KUKA KRL program: EOAChangerControl.src, EOAChangerControl.dat

--- EOAChangerControl.src ---
&ACCESS RVO4
&REL 10
&PARAM DISKPATH = KRC:\R1\TP\CNCR TP\Schunk
DEF EOAChangerControl( )

;************************************************
;              CNC Robotics Ltd
;              www.cncrobotics.co.uk
;************************************************
;     Contact: helpdesk@cncrobotics.co.uk
;     Date: 25/09/23
;     Version: 0.14.46
;************************************************
; Description: Programs for swapping the EOA tool.
;************************************************

END

GLOBAL DEF SwapTool(newTool:IN)
DECL EOA_TOOL_TYPE newTool
;HomeRobot()

HomePosition()
;WAIT FOR NOT iEOAFault
DropEOATool(ToolOnRobot)
WAIT SEC 0
nSchunkOKSwapAns = 0

WHILE nSchunkOKSwapAns<>1

MsgDialog(nSchunkOKSwapAns,"Swap the tool balance clips to the new tool","Schunk",,,,,,,"Cancel","Continue", FALSE, nSchunkMsg, E_spsMsgOpt)

ENDWHILE

PickUpEOATool(newTool)

HomePosition()
END

GLOBAL DEF DropEOATool(tool:IN)
DECL EOA_TOOL_TYPE tool

;WAIT FOR NOT iEOAFault

SWITCH tool
   CASE #SPINDLE

      IF nToolHeld <> 0 THEN
         ToolCheck()
      ELSE
         WAIT FOR (nToolHeld == 0) AND (NOT iToolLocked)
      ENDIF
      ToolRackClose()
      DropSpindle()
      bToolOnRobot = FALSE

   CASE #CEAD

      DropCead()
      bToolOnRobot = FALSE

   CASE #NONE
      EOAChangeSafe()
     ; WAIT FOR iEOALocked AND NOT iEOAUnlocked
      bToolOnRobot = FALSE
ENDSWITCH

END

GLOBAL DEF PickupEOATool(tool:IN)
DECL EOA_TOOL_TYPE tool

IF tool == #NONE THEN
   RETURN
ENDIF


EOAChangeSafe()

WAIT FOR NOT (iSpindleOnRobot OR iCeadOnRobot)

SWITCH tool
   CASE #SPINDLE
      ;Move to spindle pick position
      PickUpSpindle()
      bToolOnRobot = TRUE
   CASE #CEAD

      ;Move to Extruder pick position
      PickUpCEAD()
      ;halt
      WAIT FOR iCeadOnRobot
      IF NOT iNoEmergency THEN
         PULSE(oAckErrors,TRUE,1)
      ENDIF
      bToolOnRobot = TRUE
      ;Retract extruder from post

      ;halt
   CASE #NONE

ENDSWITCH
EOAChangeSafe()


END

GLOBAL DEF LockEOAChanger(tool:IN)
DECL EOA_TOOL_TYPE tool

WAIT FOR iAirOk

oEOAUnlock = FALSE
oEOANotLock = FALSE

WAIT FOR NOT iEOAUnlocked

IF tool <> #NONE THEN
   WAIT FOR iEOALocked
ENDIF

IF tool == #CEAD THEN
   WAIT FOR iCeadOnRobot
      IF NOT iNoEmergency THEN
         PULSE(oAckErrors,TRUE,1)
      ENDIF
ENDIF

bToolOnRobot = TRUE AND (tool <> #NONE)
toolOnRobot = tool

WAIT SEC 1

END

GLOBAL DEF UnlockEOAChanger()

WAIT FOR iAirOk

bToolOnRobot = FALSE

oEOANotLock = TRUE
oEOAUnlock = TRUE

WAIT FOR iEOAUnlocked AND NOT iEOALocked

toolOnRobot = #NONE

WAIT SEC 1

END

GLOBAL DEF SetNullTool(tool:IN)
DECL EOA_TOOL_TYPE tool

Switch tool
   CASE #SPINDLE
      BAS(#TOOL, 31)
   CASE #CEAD
      BAS(#TOOL, 32)
   CASE #NONE
      BAS(#TOOL, 0)
ENDSWITCH

END


GLOBAL DEF NullPTP(tool:IN, MoveTo:IN)
DECL EOA_TOOL_TYPE tool
DECL E6POS MoveTo

BAS(#BASE, 0)

SetNullTool(tool)


BAS(#VEL_PTP,20)


PTP MoveTo

END

GLOBAL DEFFCT BOOL CheckEOAinputs (tool:IN)
DECL EOA_TOOL_TYPE tool

SWITCH tool
CASE #SPINDLE
   RETURN iSpindleOnRobot
CASE #CEAD
   RETURN iCeadOnRobot
CASE #NONE
   RETURN NOT(iCeadOnRobot OR iSpindleOnRobot)
ENDSWITCH


ENDFCT

GLOBAL DEF CheckEOATooling(tool:IN)
DECL INT _nAns
DECL EOA_TOOL_TYPE tool

_nAns = 0

WHILE ( (CheckEOAinputs(tool)) AND (toolOnRobot<>tool) )

MsgDialog(_nAns,"Incorrect EOA tooling. Cancel program and change EOA tooling","Schunk",,,,,,,,"Cancel", FALSE, nSchunkMsg, E_spsMsgOpt)

ENDWHILE

END

--- EOAChangerControl.dat ---
&ACCESS  RV
&PARAM DISKPATH = KRC:\R1\TP\CNCR TP\Schunk
&REL 9
DEFDAT  EOACHANGERCONTROL PUBLIC

;Global Variables
GLOBAL BOOL bToolOnRobot=TRUE
GLOBAL BOOL bSchunkFault=FALSE
GLOBAL ENUM EOA_TOOL_TYPE CEAD,SPINDLE,NONE
DECL GLOBAL EOA_TOOL_TYPE toolOnRobot=#SPINDLE
GLOBAL INT nSchunkOKSwapAns=1

DECL BASIS_SUGG_T LAST_BASIS={POINT1[] "P18                     ",POINT2[] "P18                     ",CP_PARAMS[] "CPDAT18                 ",PTP_PARAMS[] "PDAT0                   ",CONT[] "                        ",CP_VEL[] "0.05                    ",PTP_VEL[] "100                     ",SYNC_PARAMS[] "SYNCDAT                 ",SPL_NAME[] "S0                      ",A_PARAMS[] "ADAT0                   "}
DECL E6POS XP1={X 2110.28467,Y 207.085190,Z 2.20077252,A 89.6821136,B 59.9209824,C 90.9203,S 22,T 59,E1 -360.000763,E2 0.0,E3 0.0,E4 0.0,E5 0.0,E6 0.0}
DECL FDAT FP1={TOOL_NO 0,BASE_NO 0,IPO_FRAME #BASE,POINT2[] " ",TQ_STATE FALSE}
DECL LDAT LCPDAT1={VEL 2.00000,ACC 100.000,APO_DIST 100.000,APO_FAC 50.0000,AXIS_VEL 100.000,AXIS_ACC 100.000,ORI_TYP #VAR,CIRC_TYP #BASE,JERK_FAC 50.0000,GEAR_JERK 50.0000,EXAX_IGN 0}
DECL E6POS XP2={X 2415.83740,Y 208.572250,Z 1.01012671,A 89.8723297,B 60.1981316,C 91.1378,S 22,T 59,E1 -360.000763,E2 0.0,E3 0.0,E4 0.0,E5 0.0,E6 0.0}
DECL FDAT FP2={TOOL_NO 0,BASE_NO 0,IPO_FRAME #BASE,POINT2[] " ",TQ_STATE FALSE}
DECL LDAT LCPDAT2={VEL 2.00000,ACC 5.00000,APO_DIST 100.000,APO_FAC 50.0000,AXIS_VEL 100.000,AXIS_ACC 100.000,ORI_TYP #VAR,CIRC_TYP #BASE,JERK_FAC 50.0000,GEAR_JERK 50.0000,EXAX_IGN 0}
DECL E6POS XP3={X 2415.85522,Y 208.560196,Z 40.6353645,A 89.8745,B 60.1985,C 91.1395645,S 22,T 59,E1 -360.000763,E2 0.0,E3 0.0,E4 0.0,E5 0.0,E6 0.0}
DECL FDAT FP3={TOOL_NO 0,BASE_NO 0,IPO_FRAME #BASE,POINT2[] " ",TQ_STATE FALSE}
DECL LDAT LCPDAT3={VEL 2.00000,ACC 5.00000,APO_DIST 100.000,APO_FAC 50.0000,AXIS_VEL 100.000,AXIS_ACC 100.000,ORI_TYP #VAR,CIRC_TYP #BASE,JERK_FAC 50.0000,GEAR_JERK 50.0000,EXAX_IGN 0}
DECL E6POS XP4={X 2116.75293,Y 208.708710,Z 41.8776550,A 89.8257751,B 60.1956673,C 91.0831833,S 22,T 59,E1 -360.000763,E2 0.0,E3 0.0,E4 0.0,E5 0.0,E6 0.0}
DECL FDAT FP4={TOOL_NO 0,BASE_NO 0,IPO_FRAME #BASE,POINT2[] " ",TQ_STATE FALSE}
DECL LDAT LCPDAT4={VEL 2.00000,ACC 5.00000,APO_DIST 100.000,APO_FAC 50.0000,AXIS_VEL 100.000,AXIS_ACC 100.000,ORI_TYP #VAR,CIRC_TYP #BASE,JERK_FAC 50.0000,GEAR_JERK 50.0000,EXAX_IGN 0}
DECL E6POS XP5={X 2110.28589,Y 207.069,Z 53.0706749,A 89.6858215,B 59.9213676,C 90.9231262,S 22,T 59,E1 -360.000763,E2 0.0,E3 0.0,E4 0.0,E5 0.0,E6 0.0}
DECL FDAT FP5={TOOL_NO 0,BASE_NO 0,IPO_FRAME #BASE,POINT2[] " ",TQ_STATE FALSE}
DECL LDAT LCPDAT5={VEL 2.00000,ACC 100.000,APO_DIST 100.000,APO_FAC 50.0000,AXIS_VEL 100.000,AXIS_ACC 100.000,ORI_TYP #VAR,CIRC_TYP #BASE,JERK_FAC 50.0000,GEAR_JERK 50.0000,EXAX_IGN 0}
DECL E6POS XP6={X 2416.12964,Y 209.042725,Z 41.9984512,A 89.6551743,B 60.2458687,C 91.1575,S 22,T 59,E1 -360.000763,E2 0.0,E3 0.0,E4 0.0,E5 0.0,E6 0.0}
DECL FDAT FP6={TOOL_NO 0,BASE_NO 0,IPO_FRAME #BASE,POINT2[] " ",TQ_STATE FALSE}
DECL LDAT LCPDAT6={VEL 2.00000,ACC 5.00000,APO_DIST 100.000,APO_FAC 50.0000,AXIS_VEL 100.000,AXIS_ACC 100.000,ORI_TYP #VAR,CIRC_TYP #BASE,JERK_FAC 50.0000,GEAR_JERK 50.0000,EXAX_IGN 0}
DECL E6POS XP7={X 2416.11230,Y 209.054535,Z 3.29431415,A 89.6530533,B 60.2455025,C 91.1557693,S 22,T 59,E1 -360.000763,E2 0.0,E3 0.0,E4 0.0,E5 0.0,E6 0.0}
DECL FDAT FP7={TOOL_NO 0,BASE_NO 0,IPO_FRAME #BASE,POINT2[] " ",TQ_STATE FALSE}
DECL LDAT LCPDAT7={VEL 2.00000,ACC 5.00000,APO_DIST 100.000,APO_FAC 50.0000,AXIS_VEL 100.000,AXIS_ACC 100.000,ORI_TYP #VAR,CIRC_TYP #BASE,JERK_FAC 50.0000,GEAR_JERK 50.0000,EXAX_IGN 0}
DECL E6POS XP8={X 2412.57593,Y 209.057129,Z 1.56290293,A 89.6524,B 60.2454529,C 91.1550293,S 22,T 59,E1 -360.000763,E2 0.0,E3 0.0,E4 0.0,E5 0.0,E6 0.0}
DECL FDAT FP8={TOOL_NO 0,BASE_NO 0,IPO_FRAME #BASE,POINT2[] " ",TQ_STATE FALSE}
DECL LDAT LCPDAT8={VEL 2.00000,ACC 5.00000,APO_DIST 100.000,APO_FAC 50.0000,AXIS_VEL 100.000,AXIS_ACC 100.000,ORI_TYP #VAR,CIRC_TYP #BASE,JERK_FAC 50.0000,GEAR_JERK 50.0000,EXAX_IGN 0}
DECL E6POS XP9={X 2225.87671,Y 209.156555,Z 2.36978531,A 89.6218,B 60.2435684,C 91.1194611,S 22,T 59,E1 -360.000763,E2 0.0,E3 0.0,E4 0.0,E5 0.0,E6 0.0}
DECL FDAT FP9={TOOL_NO 0,BASE_NO 0,IPO_FRAME #BASE,POINT2[] " ",TQ_STATE FALSE}
DECL LDAT LCPDAT9={VEL 2.00000,ACC 100.000,APO_DIST 100.000,APO_FAC 50.0000,AXIS_VEL 100.000,AXIS_ACC 100.000,ORI_TYP #VAR,CIRC_TYP #BASE,JERK_FAC 50.0000,GEAR_JERK 50.0000,EXAX_IGN 0}
DECL E6POS XP10={X 2268.25537,Y 206.572342,Z 1090.06494,A 90.2147751,B 60.5988121,C 91.2159958,S 22,T 59,E1 -360.000763,E2 0.0,E3 0.0,E4 0.0,E5 0.0,E6 0.0}
DECL FDAT FP10={TOOL_NO 0,BASE_NO 0,IPO_FRAME #BASE,POINT2[] " ",TQ_STATE FALSE}
DECL LDAT LCPDAT10={VEL 2.00000,ACC 100.000,APO_DIST 100.000,APO_FAC 50.0000,AXIS_VEL 100.000,AXIS_ACC 100.000,ORI_TYP #VAR,CIRC_TYP #BASE,JERK_FAC 50.0000,GEAR_JERK 50.0000,EXAX_IGN 0}
DECL E6POS XP11={X 2441.39771,Y 206.522354,Z 1089.56934,A 90.2275467,B 60.5963249,C 91.2292,S 22,T 59,E1 -360.000763,E2 0.0,E3 0.0,E4 0.0,E5 0.0,E6 0.0}
DECL FDAT FP11={TOOL_NO 0,BASE_NO 0,IPO_FRAME #BASE,POINT2[] " ",TQ_STATE FALSE}
DECL LDAT LCPDAT11={VEL 2.00000,ACC 5.00000,APO_DIST 100.000,APO_FAC 50.0000,AXIS_VEL 100.000,AXIS_ACC 100.000,ORI_TYP #VAR,CIRC_TYP #BASE,JERK_FAC 50.0000,GEAR_JERK 50.0000,EXAX_IGN 0}
DECL E6POS XP12={X 2441.48755,Y 206.521118,Z 1137.87341,A 90.2316818,B 60.5967445,C 91.2319260,S 22,T 59,E1 -360.000763,E2 0.0,E3 0.0,E4 0.0,E5 0.0,E6 0.0}
DECL FDAT FP12={TOOL_NO 0,BASE_NO 0,IPO_FRAME #BASE,POINT2[] " ",TQ_STATE FALSE}
DECL LDAT LCPDAT12={VEL 2.00000,ACC 5.00000,APO_DIST 100.000,APO_FAC 50.0000,AXIS_VEL 100.000,AXIS_ACC 100.000,ORI_TYP #VAR,CIRC_TYP #BASE,JERK_FAC 50.0000,GEAR_JERK 50.0000,EXAX_IGN 0}
DECL E6POS XP13={X 1809.98462,Y 206.676010,Z 1139.42065,A 90.1941833,B 60.6061363,C 91.1919708,S 22,T 59,E1 -360.000763,E2 0.0,E3 0.0,E4 0.0,E5 0.0,E6 0.0}
DECL FDAT FP13={TOOL_NO 0,BASE_NO 0,IPO_FRAME #BASE,POINT2[] " ",TQ_STATE FALSE}
DECL LDAT LCPDAT13={VEL 2.00000,ACC 100.000,APO_DIST 100.000,APO_FAC 50.0000,AXIS_VEL 100.000,AXIS_ACC 100.000,ORI_TYP #VAR,CIRC_TYP #BASE,JERK_FAC 50.0000,GEAR_JERK 50.0000,EXAX_IGN 0}
DECL E6POS XP14={X 2137.01392,Y 206.603485,Z 1138.69543,A 90.2108,B 60.6013184,C 91.2106476,S 22,T 59,E1 -360.000763,E2 0.0,E3 0.0,E4 0.0,E5 0.0,E6 0.0}
DECL FDAT FP14={TOOL_NO 0,BASE_NO 0,IPO_FRAME #BASE,POINT2[] " ",TQ_STATE FALSE}
DECL LDAT LCPDAT14={VEL 2.00000,ACC 100.000,APO_DIST 100.000,APO_FAC 50.0000,AXIS_VEL 100.000,AXIS_ACC 100.000,ORI_TYP #VAR,CIRC_TYP #BASE,JERK_FAC 50.0000,GEAR_JERK 50.0000,EXAX_IGN 0}
DECL E6POS XP15={X 2441.50073,Y 206.183929,Z 1133.35229,A 90.2278366,B 60.3237762,C 91.2293854,S 22,T 59,E1 -360.000763,E2 0.0,E3 0.0,E4 0.0,E5 0.0,E6 0.0}
DECL FDAT FP15={TOOL_NO 0,BASE_NO 0,IPO_FRAME #BASE,POINT2[] " ",TQ_STATE FALSE}
DECL LDAT LCPDAT15={VEL 2.00000,ACC 5.00000,APO_DIST 100.000,APO_FAC 50.0000,AXIS_VEL 100.000,AXIS_ACC 100.000,ORI_TYP #VAR,CIRC_TYP #BASE,JERK_FAC 50.0000,GEAR_JERK 50.0000,EXAX_IGN 0}
DECL E6POS XP16={X 2441.42163,Y 206.185043,Z 1090.78687,A 90.2242203,B 60.3234062,C 91.2270,S 22,T 59,E1 -360.000763,E2 0.0,E3 0.0,E4 0.0,E5 0.0,E6 0.0}
DECL FDAT FP16={TOOL_NO 0,BASE_NO 0,IPO_FRAME #BASE,POINT2[] " ",TQ_STATE FALSE}
DECL LDAT LCPDAT16={VEL 2.00000,ACC 5.00000,APO_DIST 100.000,APO_FAC 50.0000,AXIS_VEL 100.000,AXIS_ACC 100.000,ORI_TYP #VAR,CIRC_TYP #BASE,JERK_FAC 50.0000,GEAR_JERK 50.0000,EXAX_IGN 0}
DECL E6POS XP17={X 2436.35571,Y 206.186600,Z 1090.80188,A 90.2238159,B 60.3234825,C 91.2266083,S 22,T 59,E1 -360.000763,E2 0.0,E3 0.0,E4 0.0,E5 0.0,E6 0.0}
DECL FDAT FP17={TOOL_NO 0,BASE_NO 0,IPO_FRAME #BASE,POINT2[] " ",TQ_STATE FALSE}
DECL LDAT LCPDAT17={VEL 2.00000,ACC 5.00000,APO_DIST 100.000,APO_FAC 50.0000,AXIS_VEL 100.000,AXIS_ACC 100.000,ORI_TYP #VAR,CIRC_TYP #BASE,JERK_FAC 50.0000,GEAR_JERK 50.0000,EXAX_IGN 0}
DECL E6POS XP18={X 2248.20581,Y 206.240204,Z 1091.33704,A 90.2102356,B 60.3261757,C 91.2124405,S 22,T 59,E1 -360.000763,E2 0.0,E3 0.0,E4 0.0,E5 0.0,E6 0.0}
DECL FDAT FP18={TOOL_NO 0,BASE_NO 0,IPO_FRAME #BASE,POINT2[] " ",TQ_STATE FALSE}
DECL LDAT LCPDAT18={VEL 2.00000,ACC 100.000,APO_DIST 100.000,APO_FAC 50.0000,AXIS_VEL 100.000,AXIS_ACC 100.000,ORI_TYP #VAR,CIRC_TYP #BASE,JERK_FAC 50.0000,GEAR_JERK 50.0000,EXAX_IGN 0}
ENDDAT
